// TIA Portal project "Integration Motor Control and SCADA" (V16)

(* hardware
DEVICE "S71500/ET200MP station_1"  S7-1500 station
   slot 0: "Rail_0"  Rack  6ES7 590-1***0-0AA0
   slot 1: "PLC_1"  CPU 1511-1 PN  6ES7 511-1AK01-0AB0  V2.8
      slot 3: "CPU display_1"  6ES7591-1AA00-0AA0
      slot 32768: "PROFINET interface_1"  X1
         slot 32769: "Port_1"  X1 P1
         slot 32770: "Port_2"  X1 P2
      slot 34817: "Virtual CP interface port_1"  Virtual CP interface port  Virtual CP interface port
DEVICE "PC-System_1"  SIMATIC PC station
   slot 0: "SIMATIC PC station"  Rail  SIMATIC PC-Station  V1.0
      slot 125: "Stationmanager"  Station_Manager  V6.0.4
   slot 1: "HMI_RT_1"  WinCC RT Professional  6AV2 105-0xxxx-xxxx  16.0.0.0
*)

// ===== PLC "PLC_1"  CPU 1511-1 PN =====

VAR_GLOBAL   // PLC tag table "Default tag table"
   "LEVEL" AT %MW100 : Int;
   "Clock_Byte" AT %MB0 : Byte;
   "Clock_10Hz" AT %M0.0 : Bool;
   "Clock_5Hz" AT %M0.1 : Bool;
   "Clock_2.5Hz" AT %M0.2 : Bool;
   "Clock_2Hz" AT %M0.3 : Bool;
   "Clock_1.25Hz" AT %M0.4 : Bool;
   "Clock_1Hz" AT %M0.5 : Bool;
   "Clock_0.625Hz" AT %M0.6 : Bool;
   "Clock_0.5Hz" AT %M0.7 : Bool;
   "System_Byte" AT %MB1 : Byte;
   "FirstScan" AT %M1.0 : Bool;
   "DiagStatusUpdate" AT %M1.1 : Bool;
   "AlwaysTRUE" AT %M1.2 : Bool;
   "AlwaysFALSE" AT %M1.3 : Bool;
END_VAR

VAR_GLOBAL   // PLC tag table "Automode"
   "M_1" AT %M10.4 : Bool;
   "M_2" AT %M10.5 : Bool;
   "M_3" AT %M10.6 : Bool;
   "S0" AT %M10.7 : Bool;
   "S1" AT %M11.0 : Bool;
   "S2" AT %M11.1 : Bool;
   "S3" AT %M11.2 : Bool;
   "T00" AT %M11.3 : Bool;
   "T01" AT %M11.4 : Bool;
   "T12" AT %M11.5 : Bool;
   "T23" AT %M11.6 : Bool;
   "T31" AT %M11.7 : Bool;
   "T10" AT %M12.0 : Bool;
   "T20" AT %M12.1 : Bool;
   "T30" AT %M12.2 : Bool;
END_VAR

DATA_BLOCK "MOTOR_1"   // DB1
{ S7_Optimized_Access := 'FALSE' }
VERSION : 0.1
// stored: InstanceOfName MOTOR
"MOTOR"
BEGIN
END_DATA_BLOCK

DATA_BLOCK "MOTOR_2"   // DB2
{ S7_Optimized_Access := 'FALSE' }
VERSION : 0.1
// stored: InstanceOfName MOTOR
"MOTOR"
BEGIN
END_DATA_BLOCK

DATA_BLOCK "MOTOR_3"   // DB3
{ S7_Optimized_Access := 'FALSE' }
VERSION : 0.1
// stored: InstanceOfName MOTOR
"MOTOR"
BEGIN
END_DATA_BLOCK

DATA_BLOCK "CTRL_PANEL"   // DB6
{ S7_Optimized_Access := 'FALSE' }
VERSION : 0.1
   VAR
      START : Bool;
      STOP : Bool;
      HI : Bool;
      LO : Bool;
   END_VAR
BEGIN
END_DATA_BLOCK

// folder: System blocks/Program resources

DATA_BLOCK "T10S"   // DB5
{ S7_Optimized_Access := 'TRUE' }
AUTHOR : Simatic
FAMILY : IEC
NAME : IEC_TMR
VERSION : 1.0
// stored: InstanceOfName IEC_TIMER
"IEC_TIMER"
BEGIN
END_DATA_BLOCK

// folder: (top level)

FUNCTION_BLOCK "MOTOR"   // FB1, SCL
{ S7_Optimized_Access := 'FALSE' }
VERSION : 0.1
   VAR_INPUT
      MODE : Int;   // 1 - MAN, 2 - AUTO
      START : Bool;   // MODE = 1, START => CMD = 1
      STOP : Bool;   // MODE = 1, STOP => CMD = 0
      RUNCONDITION : Bool;   // MODE = 2, RUNCONDITION => CMD = 1
      STOPCONDITION : Bool;   // MODE = 2, STOPCONDITION => CMD = 0
      RUNFEEDBACK : Bool;
      RESET : Bool;
   END_VAR
   VAR_OUTPUT
      CMD : Bool;
      FAULT : Bool;
   END_VAR
   VAR
      DELAY_CMD : TON_TIME;
   END_VAR
BEGIN
   IF #MODE = 1 THEN
       #CMD := (#START OR #CMD) AND NOT #STOP AND NOT #FAULT;
   END_IF;

   IF #MODE = 2 THEN
       #CMD := (#RUNCONDITION OR #CMD) AND NOT #STOPCONDITION AND NOT #FAULT;
   END_IF;

   #DELAY_CMD(IN:=#CMD,
              PT:=T#5S);

   IF #DELAY_CMD.Q AND NOT #RUNFEEDBACK THEN
       #FAULT := 1;
   END_IF;

   IF #RESET THEN
       #FAULT := 0;
   END_IF;
END_FUNCTION_BLOCK

ORGANIZATION_BLOCK "Main"   // OB1, FBD, ProgramCycle
TITLE = "Main Program Sweep (Cycle)"
{ S7_Optimized_Access := 'TRUE' }
VERSION : 0.1
   VAR_INPUT
      Initial_Call : Bool;   // Initial call of this OB
      Remanence : Bool;   // =True, if remanent data are available
   END_VAR
BEGIN

REGION Network 1
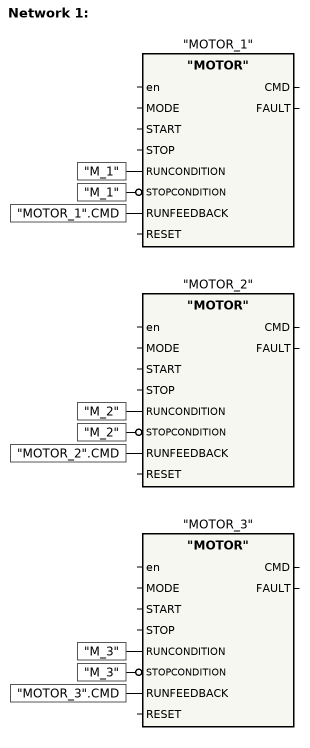
   "MOTOR_1"(RUNCONDITION := "M_1", STOPCONDITION := NOT "M_1", RUNFEEDBACK := "MOTOR_1".CMD);   // "MOTOR"
   "MOTOR_2"(RUNCONDITION := "M_2", STOPCONDITION := NOT "M_2", RUNFEEDBACK := "MOTOR_2".CMD);   // "MOTOR"
   "MOTOR_3"(RUNCONDITION := "M_3", STOPCONDITION := NOT "M_3", RUNFEEDBACK := "MOTOR_3".CMD);   // "MOTOR"
END_REGION
END_ORGANIZATION_BLOCK

ORGANIZATION_BLOCK "Sim"   // OB123, SCL, ProgramCycle
TITLE = "Main Program Sweep (Cycle)"
{ S7_Optimized_Access := 'TRUE' }
VERSION : 0.1
   VAR_INPUT
      Initial_Call : Bool;   // Initial call of this OB
      Remanence : Bool;   // =True, if remanent data are available
   END_VAR
BEGIN
   "R_TRIG_DB"(CLK:="Clock_1Hz");

   IF "MOTOR_1".RUNFEEDBACK AND "R_TRIG_DB".Q THEN
       "LEVEL" := "LEVEL" + 1;
       IF "LEVEL" >= 100 THEN
           "LEVEL" := 100;
       END_IF;
   END_IF;

   IF "MOTOR_2".RUNFEEDBACK AND "R_TRIG_DB".Q THEN
       "LEVEL" := "LEVEL" + 1;
       IF "LEVEL" >= 100 THEN
           "LEVEL" := 100;
       END_IF;
   END_IF;

   IF "MOTOR_3".RUNFEEDBACK AND "R_TRIG_DB".Q THEN
       "LEVEL" := "LEVEL" - 2;
       IF "LEVEL" <= 0 THEN
           "LEVEL" := 0;
       END_IF;
   END_IF;

   IF "LEVEL" >= 99 THEN
       "CTRL_PANEL".HI := TRUE;
   ELSE
       "CTRL_PANEL".HI := FALSE;
   END_IF;

   IF "LEVEL" <= 1 THEN
       "CTRL_PANEL".LO := TRUE;
   ELSE
       "CTRL_PANEL".LO := FALSE;
   END_IF;
END_ORGANIZATION_BLOCK

ORGANIZATION_BLOCK "AUTOMODE"   // OB124, SCL, ProgramCycle
TITLE = "Main Program Sweep (Cycle)"
{ S7_Optimized_Access := 'TRUE' }
VERSION : 0.1
   VAR_INPUT
      Initial_Call : Bool;   // Initial call of this OB
      Remanence : Bool;   // =True, if remanent data are available
   END_VAR
BEGIN
   "T10S".TON(IN:="S1",
              PT:=T#10S);

   // TRANSITION LOGICS
   "T00" := "FirstScan";
   "T01" := "S0" AND "CTRL_PANEL".START;
   "T12" := "S1" AND "T10S".Q;
   "T23" := "S2" AND "CTRL_PANEL".HI;
   "T31" := "S3" AND "CTRL_PANEL".LO;
   "T10" := "S1" AND "CTRL_PANEL".STOP;
   "T20" := "S2" AND "CTRL_PANEL".STOP;
   "T30" := "S3" AND "CTRL_PANEL".STOP;

   // STATE LOGICS
   "S0" := ("S0" OR "T00" OR "T10" OR "T20" OR "T30") AND NOT "T01";
   "S1" := ("S1" OR "T01" OR "T31") AND NOT "T12" AND NOT "T10";
   "S2" := ("S2" OR "T12") AND NOT "T23" AND NOT "T20";
   "S3" := ("S3" OR "T23") AND NOT "T31" AND NOT "T30";

   // OUTPUT LOGICS

   "M_1" := "S1" OR "S2";
   "M_2" := "S2";
   "M_3" := "S3";
END_ORGANIZATION_BLOCK

(* ===== HMI "HMI_RT_1" =====
system functions are stored by id; their names below are inferred from use
connection "Connection_1": S71200_TCP_IP, SCADA_S7_1500_OMS

HMI tags "Default tag table"
   "LEVEL" : Int AT %MW100, 500 ms
   "START" : Bool AT %DB6.DBX0.0, 500 ms
   "STOP" : Bool AT %DB6.DBX0.1, 500 ms
   "HI" : Bool AT %DB6.DBX0.2, 500 ms
   "LO" : Bool AT %DB6.DBX0.3, 500 ms
   "MOTOR_1" : 2544df81-4997-408a-afba-2450fe2ed85d AT %DB1.DBX0.0, 500 ms
   "MOTOR_2" : 2544df81-4997-408a-afba-2450fe2ed85d AT %DB2.DBX0.0, 500 ms
   "MOTOR_3" : 2544df81-4997-408a-afba-2450fe2ed85d AT %DB3.DBX0.0, 500 ms

graphic list "LIGHT": 0 'Graphic_11'; 1 'Graphic_10'

graphic list "BUTTON_GREEN": 0 'Graphic_12'; 1 'Graphic_13'

graphic list "BUTTON_RED": 0 'Graphic_7'; 1 'Graphic_8'

screen "MAIN" 1024x768
   TubePolyline "Pipe_1" at 293,520 size 190x3
   SymbolLibrary "Symbol library_2" at 203,484 size 123x85
      on Click: InvertBit("SHOW")
      Appearance <- "RUNFEEDBACK"
   TubePolyline "Pipe_2" at 295,103 size 190x3
   SymbolLibrary "Symbol library_3" at 205,67 size 123x85
      on Click: InvertBit("SHOW")
      Appearance <- "RUNFEEDBACK"
   TubePolyline "Pipe_3" at 527,481 size 190x3
   SymbolLibrary "Symbol library_1" at 389,38 size 206x557
   SymbolLibrary "Symbol library_4" at 659,438 size 123x85
      on Click: InvertBit("SHOW")
      Appearance <- "RUNFEEDBACK"
   Bar "Bar_1" at 440,54 size 100x512; MinimumValue 0; MaximumValue 100
      ProcessValue <- "LEVEL"
   GraphicIOField "Graphic I/O field_1" at 596,53 size 37x36; PictureList "LIGHT"
      ProcessValue <- "HI"
   GraphicIOField "Graphic I/O field_2" at 595,520 size 37x36; PictureList "LIGHT"
      ProcessValue <- "LO"
   GraphicIOField "Graphic I/O field_3" at 686,41 size 69x68; PictureList "BUTTON_GREEN"
      ProcessValue <- "START"
      on PressLeft: SetBit("START")
      on ReleaseLeft: ResetBit("START")
   GraphicIOField "Graphic I/O field_4" at 765,47 size 69x68; PictureList "BUTTON_RED"
      on ReleaseLeft: ResetBit("STOP")
      on PressLeft: SetBit("STOP")
      ProcessValue <- "STOP"
   ScreenWindow "Screen window_2" at 101,358 size 150x300; ScreenName "MOTOR"
      Visibility <- "SHOW"
   ScreenWindow "Screen window_1" at 52,0 size 150x300; ScreenName "MOTOR"
      Visibility <- "SHOW"
   ScreenWindow "Screen window_3" at 783,201 size 150x300; ScreenName "MOTOR"
      Visibility <- "SHOW"

screen "MOTOR" 140x290
   ComboBox "Combo box_1" at 20,41 size 109x30; Text1 'AUTO'; Text0 'MAN'
      SelectedIndex <- ".MODE"
   Button "Button_1" at 22,84 size 107x30; TextOff 'START'
      on PressLeft: SetBit(".START")
      on ReleaseLeft: ResetBit(".START")
   Button "Button_2" at 20,135 size 107x30; TextOff 'STOP'
      on PressLeft: SetBit(".STOP")
      on ReleaseLeft: ResetBit(".STOP")
   Circle "Circle_1" at 26,173 size 62x62
      Appearance <- ".RUNFEEDBACK"
   Circle "Circle_2" at 75,211 size 24x24
      Appearance <- ".FAULT"
   Button "Button_3" at 20,249 size 107x30; TextOff 'RESET'
      on PressLeft: SetBit(".RESET")
      on ReleaseLeft: ResetBit(".RESET")
   GraphicView "Graphic view_1" at 111,3 size 26x22; Picture "Graphic_14"
      on Click: ResetBit(".SHOW")
*)